{attribute 'linkalways'} 
{attribute 'no_explicit_call' := 'This FB is a CLASS and must be accessed using methods or properties'}
{attribute 'enable_dynamic_creation'}
FUNCTION_BLOCK Node_F_VN_FillRotatedRectangle EXTENDS VisionNode
VAR
    stRectangle : _TcVnRotatedRectangle;
    ipDestImage : _ITcVnImage;
    aColor : _TcVnVector4_LREAL;
    hrPrev : _HRESULT(S_OK);
	hresult : _HRESULT(S_OK);
END_VAR

METHOD PUBLIC  Clone : I_Node
VAR
	pNode : POINTER TO Node_F_VN_FillRotatedRectangle;
END_VAR
pNode := __NEW(Node_F_VN_FillRotatedRectangle);
Clone := pNode^;
END_METHOD

METHOD FB_init : BOOL
VAR_INPUT
	bInitRetains : BOOL; // if TRUE, the retain variables are initialized (warm start / cold start)
	bInCopyCode : BOOL;  // if TRUE, the instance afterwards gets moved into the copy code (online change)
END_VAR
AddInput('stRectangle', stRectangle);
AddInput('ipDestImage', ipDestImage);
AddInput('aColor', aColor);
AddInput('hrPrev', hrPrev);
AddOutput('ipDestImage', ipDestImage);
AddOutput('hresult',hresult);
END_METHOD

METHOD PROTECTED  OnExecute : HRESULT
hresult.Value := F_VN_FillRotatedRectangle(
    stRectangle := stRectangle.Value,
	ipDestImage := ipDestImage.Value,
    aColor := aColor.Value,
	hrPrev:= hrPrev.Value);
END_METHOD

METHOD PUBLIC PreExecutionCheck
VAR_INPUT
	Check : I_PreExecutionChecks;
END_VAR
Check.IsTrue(ipDestImage.IsValid, 'ipDestImage must contain an image');
END_METHOD

END_FUNCTION_BLOCK

(* stored: Version 1.1.0.1, ProductVersion 3.1.4024.13
   POU Node_F_VN_FillRotatedRectangle: Id {ba0c456d-58da-0017-179e-c007f52c8878}, SpecialFunc None
   Folder Constructor: Id {a8180801-fbf9-07cb-2316-352617ecb1cc}
   Method Clone: Id {64235ec6-56f5-06be-2405-15ba6ab98c6d}
   Method FB_init: Id {ab4868f5-2375-0f70-3fe7-020bb6c11621}
   Method OnExecute: Id {1bd06e1a-fe44-0f50-0cf8-070f075c3788}
   Method PreExecutionCheck: Id {a8aafcfd-321a-0a03-3125-9d94bf7df0a3} *)
